% RSLogix 500 project Betriebsstundenzähler.RSS, saved by version 8.30.00.16 %
PROJECT "UNTITLED"    % processor: Bul.1763 MicroLogix 1100 Series B %

PROGRAM FILES
  LAD 2   12 rungs

DATA FILES
  O0 OUTPUT  4 elements
  I1 INPUT  6 elements
  S2 STATUS  66 elements
  B3 BINARY  1 elements
  T4 TIMER  1 elements
  C5 COUNTER  4 elements
  R6 CONTROL  1 elements
  N7 INTEGER  4 elements
  F8 FLOAT  1 elements

LADDER 2
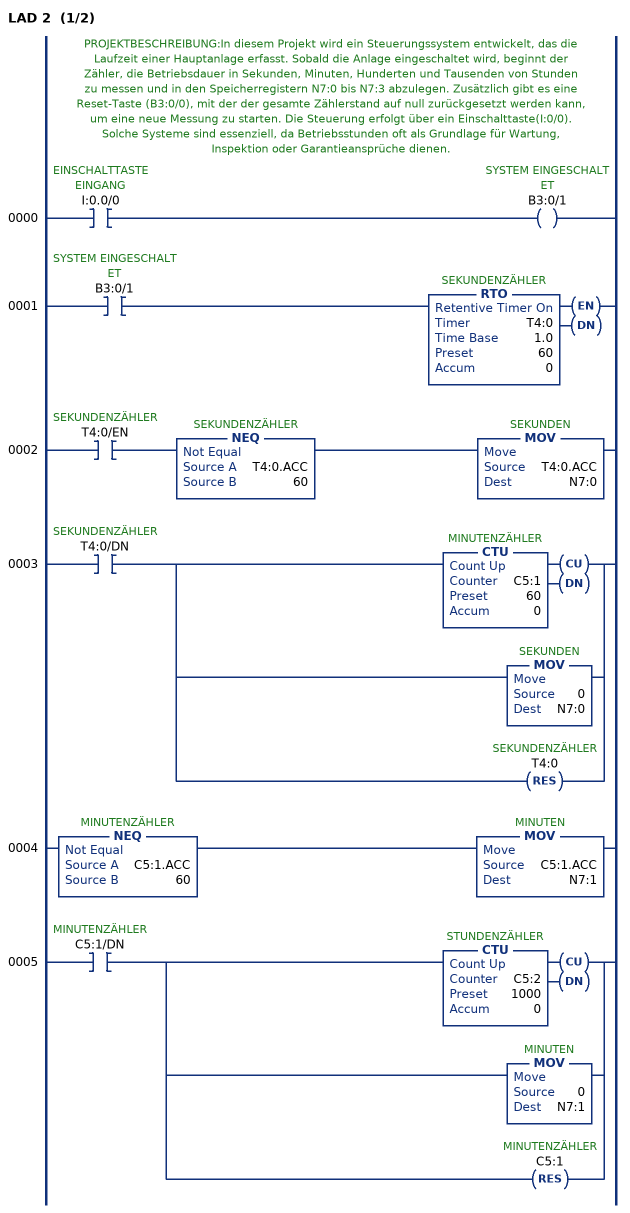
% Rung: 0 %
% PROJEKTBESCHREIBUNG:In diesem Projekt wird ein Steuerungssystem entwickelt, das die Laufzeit einer Hauptanlage erfasst. Sobald die Anlage eingeschaltet wird, beginnt der Zähler, die Betriebsdauer in Sekunden, Minuten, Hunderten und Tausenden von Stunden zu messen und in den Speicherregistern N7:0 bis N7:3 abzulegen. Zusätzlich gibt es eine Reset-Taste (B3:0/0), mit der der gesamte Zählerstand auf null zurückgesetzt werden kann, um eine neue Messung zu starten. Die Steuerung erfolgt über ein Einschalttaste(I:0/0). Solche Systeme sind essenziell, da Betriebsstunden oft als Grundlage für Wartung, Inspektion oder Garantieansprüche dienen. %
SOR XIC I:0.0/0 OTE B3:0/1 EOR
%   I:0.0/0  "EINSCHALTTASTE EINGANG" %
%   B3:0/1  "SYSTEM EINGESCHALTET" %
% Rung: 1 %
SOR XIC B3:0/1 RTO T4:0 1.0 60 0 EOR
%   B3:0/1  "SYSTEM EINGESCHALTET" %
%   T4:0  "SEKUNDENZÄHLER" %
% Rung: 2 %
SOR XIC T4:0/EN NEQ T4:0.ACC 60 MOV T4:0.ACC N7:0 EOR
%   T4:0  "SEKUNDENZÄHLER" %
%   N7:0  "SEKUNDEN" %
% Rung: 3 %
SOR XIC T4:0/DN BST CTU C5:1 60 0 NXB MOV 0 N7:0 NXB RES T4:0 BND EOR
%   T4:0  "SEKUNDENZÄHLER" %
%   C5:1  "MINUTENZÄHLER" %
%   N7:0  "SEKUNDEN" %
% Rung: 4 %
SOR NEQ C5:1.ACC 60 MOV C5:1.ACC N7:1 EOR
%   C5:1  "MINUTENZÄHLER" %
%   N7:1  "MINUTEN" %
% Rung: 5 %
SOR XIC C5:1/DN BST CTU C5:2 1000 0 NXB MOV 0 N7:1 NXB RES C5:1 BND EOR
%   C5:1  "MINUTENZÄHLER" %
%   C5:2  "STUNDENZÄHLER" %
%   N7:1  "MINUTEN" %

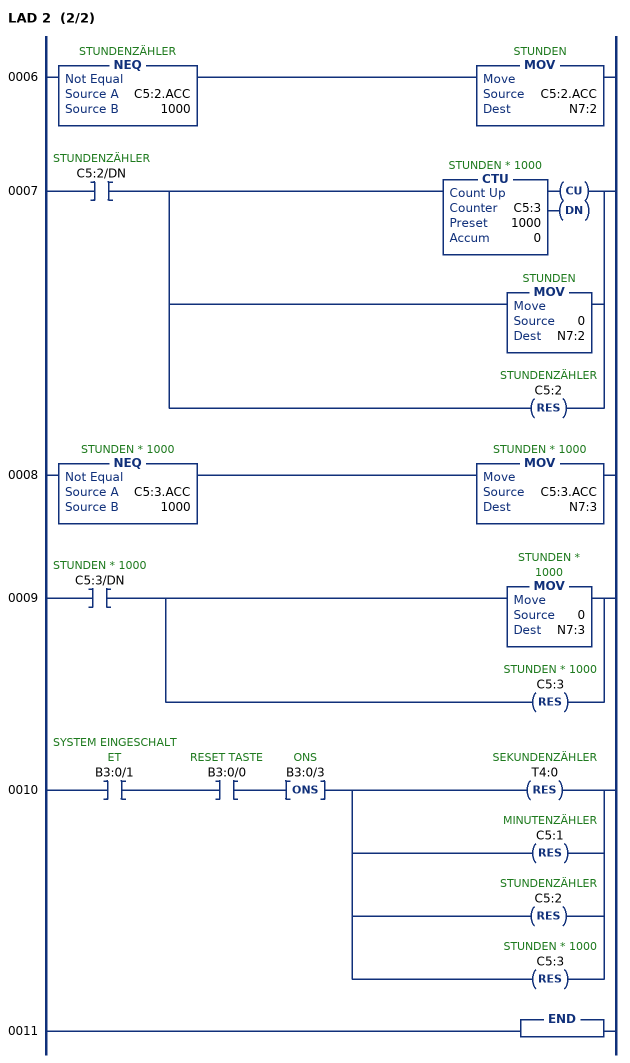
% Rung: 6 %
SOR NEQ C5:2.ACC 1000 MOV C5:2.ACC N7:2 EOR
%   C5:2  "STUNDENZÄHLER" %
%   N7:2  "STUNDEN" %
% Rung: 7 %
SOR XIC C5:2/DN BST CTU C5:3 1000 0 NXB MOV 0 N7:2 NXB RES C5:2 BND EOR
%   C5:2  "STUNDENZÄHLER" %
%   C5:3  "STUNDEN * 1000" %
%   N7:2  "STUNDEN" %
% Rung: 8 %
SOR NEQ C5:3.ACC 1000 MOV C5:3.ACC N7:3 EOR
%   C5:3  "STUNDEN * 1000" %
%   N7:3  "STUNDEN * 1000" %
% Rung: 9 %
SOR XIC C5:3/DN BST MOV 0 N7:3 NXB RES C5:3 BND EOR
%   C5:3  "STUNDEN * 1000" %
%   N7:3  "STUNDEN * 1000" %
% Rung: 10 %
SOR XIC B3:0/1 XIC B3:0/0 ONS B3:0/3 BST RES T4:0 NXB RES C5:1 NXB RES C5:2 NXB RES C5:3 BND EOR
%   B3:0/1  "SYSTEM EINGESCHALTET" %
%   B3:0/0  "RESET TASTE" %
%   B3:0/3  "ONS" %
%   T4:0  "SEKUNDENZÄHLER" %
%   C5:1  "MINUTENZÄHLER" %
%   C5:2  "STUNDENZÄHLER" %
%   C5:3  "STUNDEN * 1000" %
% Rung: 11 %
SOR END EOR

OTHER DOCUMENTED ADDRESSES
  B3:0/2  "ONS"
  C4:0  "SEKUNDENZÄHLER"
  C5:0  "SEKUNDENZÄHLER"

DATA TABLE (non-zero values as saved)
DATA T4
% .PRE .ACC %
% T4:0 % 60 0
DATA C5
% .PRE .ACC %
% C5:0 % 60 0
% C5:1 % 60 0
% C5:2 % 1000 0
% C5:3 % 1000 0
